FUNCTION_BLOCK Actuator_Fault_CAT (* Composite Function Block Type *)
  (* Standard: 61499-2 *)
  (* Version 0.0, 2/24/2026, Schneider Electric, template *)
  PACKAGE Main;
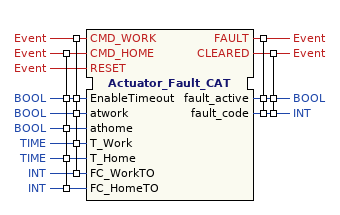
  EVENT_INPUT
    CMD_WORK WITH EnableTimeout, atwork, T_Work, FC_WorkTO; (* Initialization Request *)
    CMD_HOME WITH EnableTimeout, athome, T_Home, FC_HomeTO; (* Normal Execution Request *)
    RESET;
  END_EVENT
  EVENT_OUTPUT
    FAULT WITH fault_active, fault_code; (* Initialization Confirm *)
    CLEARED WITH fault_active, fault_code; (* Execution Confirmation *)
  END_EVENT
  VAR_INPUT
    EnableTimeout : BOOL; (* Input event qualifier *)
    atwork : BOOL;
    athome : BOOL;
    T_Work : TIME;
    T_Home : TIME;
    FC_WorkTO : INT;
    FC_HomeTO : INT;
  END_VAR
  VAR_OUTPUT
    fault_active : BOOL; (* Output event qualifier *)
    fault_code : INT;
  END_VAR
  (* WorkTimeout *)
  (* Home Timeout *)
  (* Memory of Fault *)
  FBS
    ED_Work : E_DELAY;
    ED_Home : E_DELAY;
    GateStartWork : E_SWITCH;
    GateStartHome : E_SWITCH;
    WorkTimeoutCheck : E_SWITCH;
    HomeTimeoutChceck : E_SWITCH;
    NOT_Fault : NOT_12669C4E53BA46410; {SET_ATTRIBUTE(Configuration.GenericFBType.InterfaceParams, Runtime.Standard#CNT:=1)}
    NOT_AtWork : NOT_12669C4E53BA46410; {SET_ATTRIBUTE(Configuration.GenericFBType.InterfaceParams, Runtime.Standard#CNT:=1)}
    NOT_AtHome : NOT_12669C4E53BA46410; {SET_ATTRIBUTE(Configuration.GenericFBType.InterfaceParams, Runtime.Standard#CNT:=1)}
    AND_StartWork : AND_148CCC6046D4CE74C; {SET_ATTRIBUTE(Configuration.GenericFBType.InterfaceParams, Runtime.Standard#CNT:=2)}
    AND_StartHome : AND_148CCC6046D4CE74C; {SET_ATTRIBUTE(Configuration.GenericFBType.InterfaceParams, Runtime.Standard#CNT:=2)}
    Latch : FaultLatch;
  END_FBS
  EVENT_CONNECTIONS
    GateStartWork.EO1 TO ED_Work.START;
    WorkTimeoutCheck.EO1 TO Latch.SET_WORK;
    GateStartHome.EO1 TO ED_Home.START;
    Latch.FAULT TO FAULT;
    Latch.CLEARED TO CLEARED;
    RESET TO Latch.RESET;
    ED_Work.EO TO NOT_AtWork.REQ;
    NOT_AtWork.CNF TO WorkTimeoutCheck.EI;
    CMD_WORK TO NOT_Fault.REQ;
    AND_StartWork.CNF TO GateStartWork.EI;
    NOT_Fault.CNF TO AND_StartWork.REQ;
    ED_Home.EO TO NOT_AtHome.REQ;
    AND_StartHome.CNF TO GateStartHome.EI;
    NOT_AtHome.CNF TO HomeTimeoutChceck.EI;
    HomeTimeoutChceck.EO1 TO Latch.SET_HOME;
    CMD_HOME TO AND_StartHome.REQ;
  END_CONNECTIONS
  DATA_CONNECTIONS
    Latch.fault_active TO NOT_Fault.IN1;
    AND_StartWork.OUT TO GateStartWork.G;
    T_Work TO ED_Work.DT;
    atwork TO NOT_AtWork.IN1;
    NOT_AtWork.OUT1 TO WorkTimeoutCheck.G;
    AND_StartHome.OUT TO GateStartHome.G;
    T_Home TO ED_Home.DT;
    athome TO NOT_AtHome.IN1;
    NOT_AtHome.OUT1 TO HomeTimeoutChceck.G;
    Latch.fault_active TO fault_active;
    Latch.fault_code TO fault_code;
    FC_WorkTO TO Latch.FC_WorkTO;
    FC_HomeTO TO Latch.FC_HomeTO;
    NOT_Fault.OUT1 TO AND_StartWork.IN1;
    EnableTimeout TO AND_StartWork.IN2;
    NOT_Fault.OUT1 TO AND_StartHome.IN1;
    EnableTimeout TO AND_StartHome.IN2;
  END_CONNECTIONS
END_FUNCTION_BLOCK
